FUNCTION isVentilOpen : BOOL
VAR_INPUT
	pd 		: REFERENCE TO ST_ProcessData;
END_VAR
VAR
END_VAR

isVentilOpen := pd.incident.incidentWaterFlow;

END_FUNCTION

(* stored: Version 1.1.0.1
   POU isVentilOpen: Id {14b65eaf-864a-4731-8613-d210785d0b89}, SpecialFunc None *)
